// Mitsubishi GX Works2 project: function_block   PLC: Q03UDV
// turma1

// task Task_01 (event TRUE, interval 0, priority 31): POU_01
// task ST_Example (event TRUE, interval 0, priority 31): ST_Example

PROGRAM POU_01
VAR
  CTD_1 : CTD;
  CTU_2 : CTU;
  CTUD_1 : CTUD;
  fbContadorDeProcessos2 : CTUD;
  TP_1 : TP;
  TOF_1 : TOF;
  TON_1 : TON;
  TimeTP : TIME;
  TimeON : TIME;
  TimeOFF : TIME;
  dr : TIME;
  TP_2 : TP;
  TP_3 : TP;
  TOF_2 : TOF;
  TON_2 : TON;
  TPtimer : TIME;
  TONtimer : TIME;
  TOFtimer : TIME;
  TON_3 : TON;
  TON2timer : TIME;
  fbBlinker_1 : fbBlinker;
  result : DWORD;
  resu : DWORD;
  resultado : DWORD;
  final : DWORD;
  iOperador : STRING[32];
  estrutura_op : INT;
  iHabilitar : BOOL;
  i_Valor1 : INT;
  i_Valor2 : INT;
END_VAR
(* structured ladder/FBD written out as ST: instructions are called as NAME(EN, inputs, outputs); _pN, _eN, _tN stand for wires *)
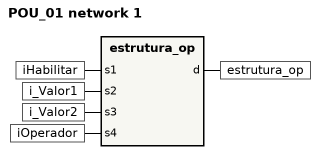
(* network 1 *)
estrutura_op := estrutura_op(iHabilitar, i_Valor1, i_Valor2, iOperador);
END_PROGRAM

FUNCTION fun_Soma_int
VAR_INPUT
  i_xHabilitar : BOOL;
  i_iElemento1 : INT;
  i_iElemento2 : INT;
END_VAR
(* structured ladder/FBD written out as ST: instructions are called as NAME(EN, inputs, outputs); _pN, _eN, _tN stand for wires *)
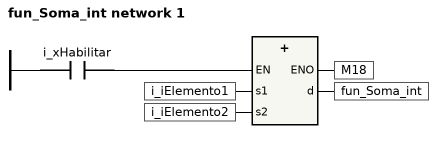
(* network 1 *)
_e1 := +(i_xHabilitar, i_iElemento1, i_iElemento2, fun_Soma_int);
M18 := _e1;
END_FUNCTION

FUNCTION fun_SubInteiro
VAR_INPUT
  i_xHabilitar2 : BOOL;
  i_iElemento3 : INT;
  i_iElemento4 : INT;
END_VAR
(* structured ladder/FBD written out as ST: instructions are called as NAME(EN, inputs, outputs); _pN, _eN, _tN stand for wires *)
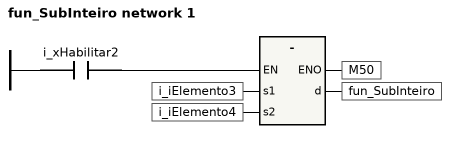
(* network 1 *)
_e1 := -(i_xHabilitar2, i_iElemento3, i_iElemento4, fun_SubInteiro);
M50 := _e1;
END_FUNCTION

FUNCTION fun_Mult_Int
VAR_INPUT
  i_xHabilitar3 : BOOL;
  i_iElemento4 : INT;
  i_iElemento5 : INT;
END_VAR
(* structured ladder/FBD written out as ST: instructions are called as NAME(EN, inputs, outputs); _pN, _eN, _tN stand for wires *)
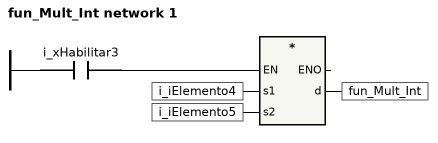
(* network 1 *)
*(i_xHabilitar3, i_iElemento4, i_iElemento5, fun_Mult_Int);
END_FUNCTION

FUNCTION_BLOCK fbBlinker
VAR_INPUT
  i_xEnable : BOOL;
  i_tHighPulse : TIME;
  i_tLowPulse : TIME;
END_VAR
VAR_OUTPUT
  o_xPulse : BOOL;
END_VAR
VAR
  fbTimerHigh : TP;
  fbTimerLow : TOF;
  auxiliar : BOOL;
  TP_1 : TP;
  TOF_1 : TOF;
END_VAR
(* structured ladder/FBD written out as ST: instructions are called as NAME(EN, inputs, outputs); _pN, _eN, _tN stand for wires *)
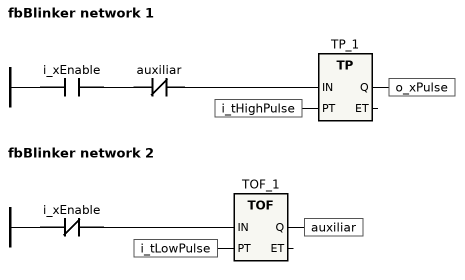
(* network 1 *)
TP_1(IN := i_xEnable AND NOT auxiliar, PT := i_tHighPulse, Q => o_xPulse);
(* network 2 *)
TOF_1(IN := NOT i_xEnable, PT := i_tLowPulse, Q => auxiliar);
END_FUNCTION_BLOCK

FUNCTION_BLOCK Operacoes
VAR_INPUT
  i_Enable1 : BOOL;
  i_Enable2 : BOOL;
END_VAR
END_FUNCTION_BLOCK

PROGRAM ST_Example
VAR
  iDR : ARRAY [0..9] OF INT;  (* declaração de variavel ST *)
END_VAR
VAR CONSTANT
  iEle01 : INT := 15;  (* elemento 01 de operação *)
  iEle02 : INT := 5;  (* elemento 02 de operação *)
END_VAR
VAR
  fbBlinkerTestST : fbBlinker;  (* declaração de variavel ST *)
  fbTPTestST : TP;  (* declaração de variavel ST *)
  x_starblink : TP;  (* declaração de variavel ST *)
  x_pulseStarblink : TP;  (* declaração de variavel ST *)
  xTesteOperacao : ARRAY [0..9] OF INT;  (* declaração de variavel ST *)
  iHabilitar : INT;
  resultado : INT;
  StringResult : STRING[32];
  resultado2 : INT;
  StringResult2 : STRING[32];
END_VAR

iDR[0] := iEle01 + iEle02;
iDR[1] := iEle01 - iEle02;
iDR[2] := iEle01 + iEle02;
iDR[3] := iEle01 / iEle02;
iDR[4] := iEle01 MOD iEle02;
(*iDR[3] := MOD(iEle01,  iEle02);*)

fbBlinkerTestST(i_xEnable:= M1010 , i_tHighPulse:= T#2s, i_tLowPulse:= T#500ms ,o_xPulse:= Y1010);
(*fbTPTestST(IN:= ?BOOL? ,PT:= ?TIME? ,Q:= ?BOOL? ,ET:= ?TIME? );*)
(*ENO := MOD(M55, iEle01, iEle02, D27)*)

iDR[5] := fbSoma( 10 , 10);
iDR[6] := fun_subtracao( 15 , 10);
iDR[7] := funMultiplicacao( 5 , 2);
iDR[8] := funDIV( 10 , 2);

(****************************************************************************************************)

resultado := estrutura_op( M0 , k10 , k10 , StringResult);
END_PROGRAM

FUNCTION fbSoma
VAR_INPUT
  i_num1 : INT;
  i_num2 : INT;
END_VAR

fbSoma := i_num1 + i_num2;
END_FUNCTION

FUNCTION fun_subtracao
VAR_INPUT
  i_num3 : INT;
  i_num4 : INT;
END_VAR
fun_subtracao := i_num3 - i_num4;
END_FUNCTION

FUNCTION funMultiplicacao
VAR_INPUT
  i_num5 : INT;
  i_num6 : INT;
END_VAR
funMultiplicacao := i_num5 * i_num6;
END_FUNCTION

FUNCTION funDIV
VAR_INPUT
  i_num7 : INT;
  i_num8 : INT;
END_VAR
funDIV := i_num7 / i_num8;
END_FUNCTION

FUNCTION_BLOCK fboperacoes
VAR CONSTANT
  i_nume : INT := 5;
  i_nume : INT := 5;
END_VAR

END_FUNCTION_BLOCK

FUNCTION estrutura_op
VAR_INPUT
  iHabilitar : BOOL;
  i_Valor1 : INT;
  i_Valor2 : INT;
  iOperador : STRING[32];
END_VAR
IF iHabilitar THEN 
	IF iOperador = "+" THEN
					estrutura_op:= i_Valor1 + i_Valor2;
		ELSIF iOperador = "-" THEN 
					estrutura_op := i_Valor1 - i_Valor2;
		ELSIF iOperador = "*" THEN 
					estrutura_op:= i_Valor1 * i_Valor2;		
		ELSIF iOperador = "/" THEN 
					estrutura_op := i_Valor1 / i_Valor2;
		ELSE 
					estrutura_op:= 32767;
	END_IF;
END_IF;
END_FUNCTION

FUNCTION Estrututa_Case
VAR_INPUT
  iHabilitar1 : INT;
  i_Valor3 : INT;
  i_Valor4 : INT;
  iOperador1 : STRING[32];
END_VAR
VAR
  aux : INT;
  auxiliar : INT;
END_VAR

END_FUNCTION
